FUNCTION_BLOCK RingTokenMember (* Basic Function Block Type *)
  (* Standard: 61499-2 *)
  (* Version 0.2, 2003-12-04, JHC, Rockwell Automation, Renamed for better indexing. *)
  (* Version 0.1, 2002-11-05, JHC, Rockwell Automation, Corrected missing ST element in Algorithm REQ. *)
  (* Version 0.0, 2000-05-30, JHC, Rockwell Automation *)
  (* Compiler header: package fb.rt.template; *)
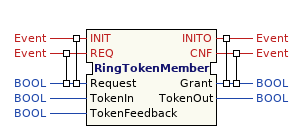
  EVENT_INPUT
    INIT WITH Request; (* Initialization Request *)
    REQ WITH Request; (* Normal Execution Request *)
  END_EVENT
  EVENT_OUTPUT
    INITO WITH Grant; (* Initialization Confirm *)
    CNF WITH Grant; (* Execution Confirmation *)
  END_EVENT
  VAR_INPUT
    Request : BOOL; (* Input event qualifier *)
    TokenIn : BOOL;
    TokenFeedback : BOOL;
  END_VAR
  VAR_OUTPUT
    Grant : BOOL; (* Output event qualifier *)
    TokenOut : BOOL;
  END_VAR
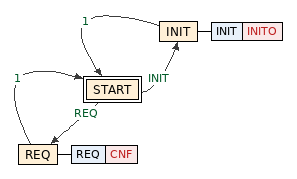
  EC_STATES
    START; (* Initial State *)
    INIT : INIT -> INITO; (* Initialization *)
    REQ : REQ -> CNF; (* Normal execution *)
  END_STATES
  EC_TRANSITIONS
    START TO INIT := INIT;
    INIT TO START := 1;
    START TO REQ := REQ;
    REQ TO START := 1;
  END_TRANSITIONS
  ALGORITHM INIT IN ST: (* Initialization algorithm *)
Grant := FALSE;
  END_ALGORITHM
  ALGORITHM REQ IN Java: (* Normally executed algorithm *)
if(TokenFeedback.value) {
	TokenOut.value = true;
	Grant.value = false;
}
else {
	if(TokenIn.value) {
		if(Request.value) {
			Grant.value = true;
			TokenOut.value = false;
		}
		else {
			Grant.value = false;
			TokenOut.value = true;
		}
	}
	else {
		TokenOut.value = false;
		Grant.value = false;
	}
}
  END_ALGORITHM
END_FUNCTION_BLOCK
